{attribute 'TcGenerated'}
// This function has been automatically generated from the project information.
VAR_GLOBAL CONSTANT
    {attribute 'const_non_replaced'}
    {attribute 'linkalways'}
    stLibVersion_plc_kfe_rix_vac : ST_LibVersion := (iMajor := 2, iMinor := 0, iBuild := 0, iRevision := 0, sVersion := '2.0.0');
END_VAR

(* stored: Version 1.1.0.1, ProductVersion 3.1.4024.6
   GVL Global_Version: Id 3d0d148e-a39a-437b-950c-3801a288457f *)
